Fanuc KAREL source: VT_DELETE_PQ.kl

PROGRAM T
%NOLOCKGROUP
VAR
 v0 : INTEGER
 v1 : INTEGER
 v2 : INTEGER
BEGIN
 VT_DELETE_PQ(v0, v1, v2)
END T
